FUNCTION_BLOCK PowerTask EXTENDS MotionTask IMPLEMENTS I_MotionPowerTask
VAR
	McPower : MC_Power;
	{attribute 'hide'}
	_InhibitFeedForward : BOOL;
	{attribute 'hide'}
	_InhibitFeedBackward : BOOL;
END_VAR

{attribute 'monitoring' := 'call'}
PROPERTY Busy : BOOL
GET
Busy := FALSE; (*MC Power Busy behaves busy as long as enabled*)
END_GET
END_PROPERTY

METHOD CyclicLogic
McPower(Axis := _Axis.Axis, Enable_Positive := NOT _InhibitFeedForward, Enable_Negative := NOT _InhibitFeedBackward);
END_METHOD

METHOD Disable
McPower.Enable := FALSE;
END_METHOD

METHOD Enable
McPower.Enable := TRUE;
END_METHOD

{attribute 'monitoring' := 'call'}
PROPERTY Enabled : BOOL
GET
Enabled := McPower.Status;
END_GET
END_PROPERTY

{attribute 'monitoring' := 'call'}
PROPERTY Error : BOOL
GET
Error := McPower.Error;
END_GET
END_PROPERTY

{attribute 'monitoring' := 'call'}
PROPERTY ErrorId : UDINT
GET
ErrorId := McPower.ErrorID;
END_GET
END_PROPERTY

METHOD Execute : BOOL
Execute := TRUE;
END_METHOD

{attribute 'monitoring' := 'call'}
PROPERTY InhibitFeedBackward : BOOL
GET
InhibitFeedBackward := _InhibitFeedBackward;
END_GET
SET
_InhibitFeedBackward := InhibitFeedBackward;
END_SET
END_PROPERTY

{attribute 'monitoring' := 'call'}
PROPERTY InhibitFeedForward : BOOL
GET
InhibitFeedForward := _InhibitFeedForward;
END_GET
SET
_InhibitFeedForward := InhibitFeedForward;
END_SET
END_PROPERTY

{attribute 'monitoring' := 'call'}
PROPERTY Override : LREAL
SET
McPower.Override := Override;
END_SET
END_PROPERTY

END_FUNCTION_BLOCK

(* stored: Version 1.1.0.1, ProductVersion 3.1.4026.18
   POU PowerTask: Id {b7f8a915-7c01-4597-bf81-b5270bb601ec}, SpecialFunc None
   Property Busy: Id {afb70197-5866-4b24-aa82-ff97fa7e1a58}
   Get Get: Id {b9ea71e0-a830-460c-a3a1-a993960f89ca}
   Method CyclicLogic: Id {cfe78734-3b00-4683-82a1-1ac563d2b02a}
   Method Disable: Id {4bd23167-cd30-4dc4-a52d-e1468c5ca63d}
   Method Enable: Id {ae7c6175-803b-4126-a0ba-33b30c6b3a88}
   Property Enabled: Id {d753b03b-686b-4ec9-b808-6930e87c14a6}
   Get Get: Id {4c3a00b4-4a7b-4b28-ab83-e9aaa3d61857}
   Property Error: Id {aa6b8469-574c-4131-a79f-e13bc0ffa735}
   Get Get: Id {11c79cf6-5769-4090-a02e-82566b4115d3}
   Property ErrorId: Id {b02694bf-0077-4347-8c62-166896b8399f}
   Get Get: Id {1134fcce-2208-4029-84c0-5ef0353ecc87}
   Method Execute: Id {f6731706-bd10-4512-91cf-c4fab51a2576}
   Property InhibitFeedBackward: Id {b13b115e-9a71-4a6b-8cb2-6051623dbcee}
   Get Get: Id {cedd79f4-bbed-4f2e-90c8-17d66c596319}
   Set Set: Id {dc06493c-7e8f-4d12-8386-01bfd4fbf75e}
   Property InhibitFeedForward: Id {f3bb0628-6869-4954-8f3e-aa14dd593620}
   Get Get: Id {ea17edd2-e9f9-45ab-818c-bb3d1ecabde7}
   Set Set: Id {c7f79851-16a7-488a-9224-359994080505}
   Property Override: Id {21edb0d4-9eb0-414a-b8f2-ad2f4009995b}
   Set Set: Id {ecae7212-8297-4cd4-9cd1-a1cd5e57026f} *)
